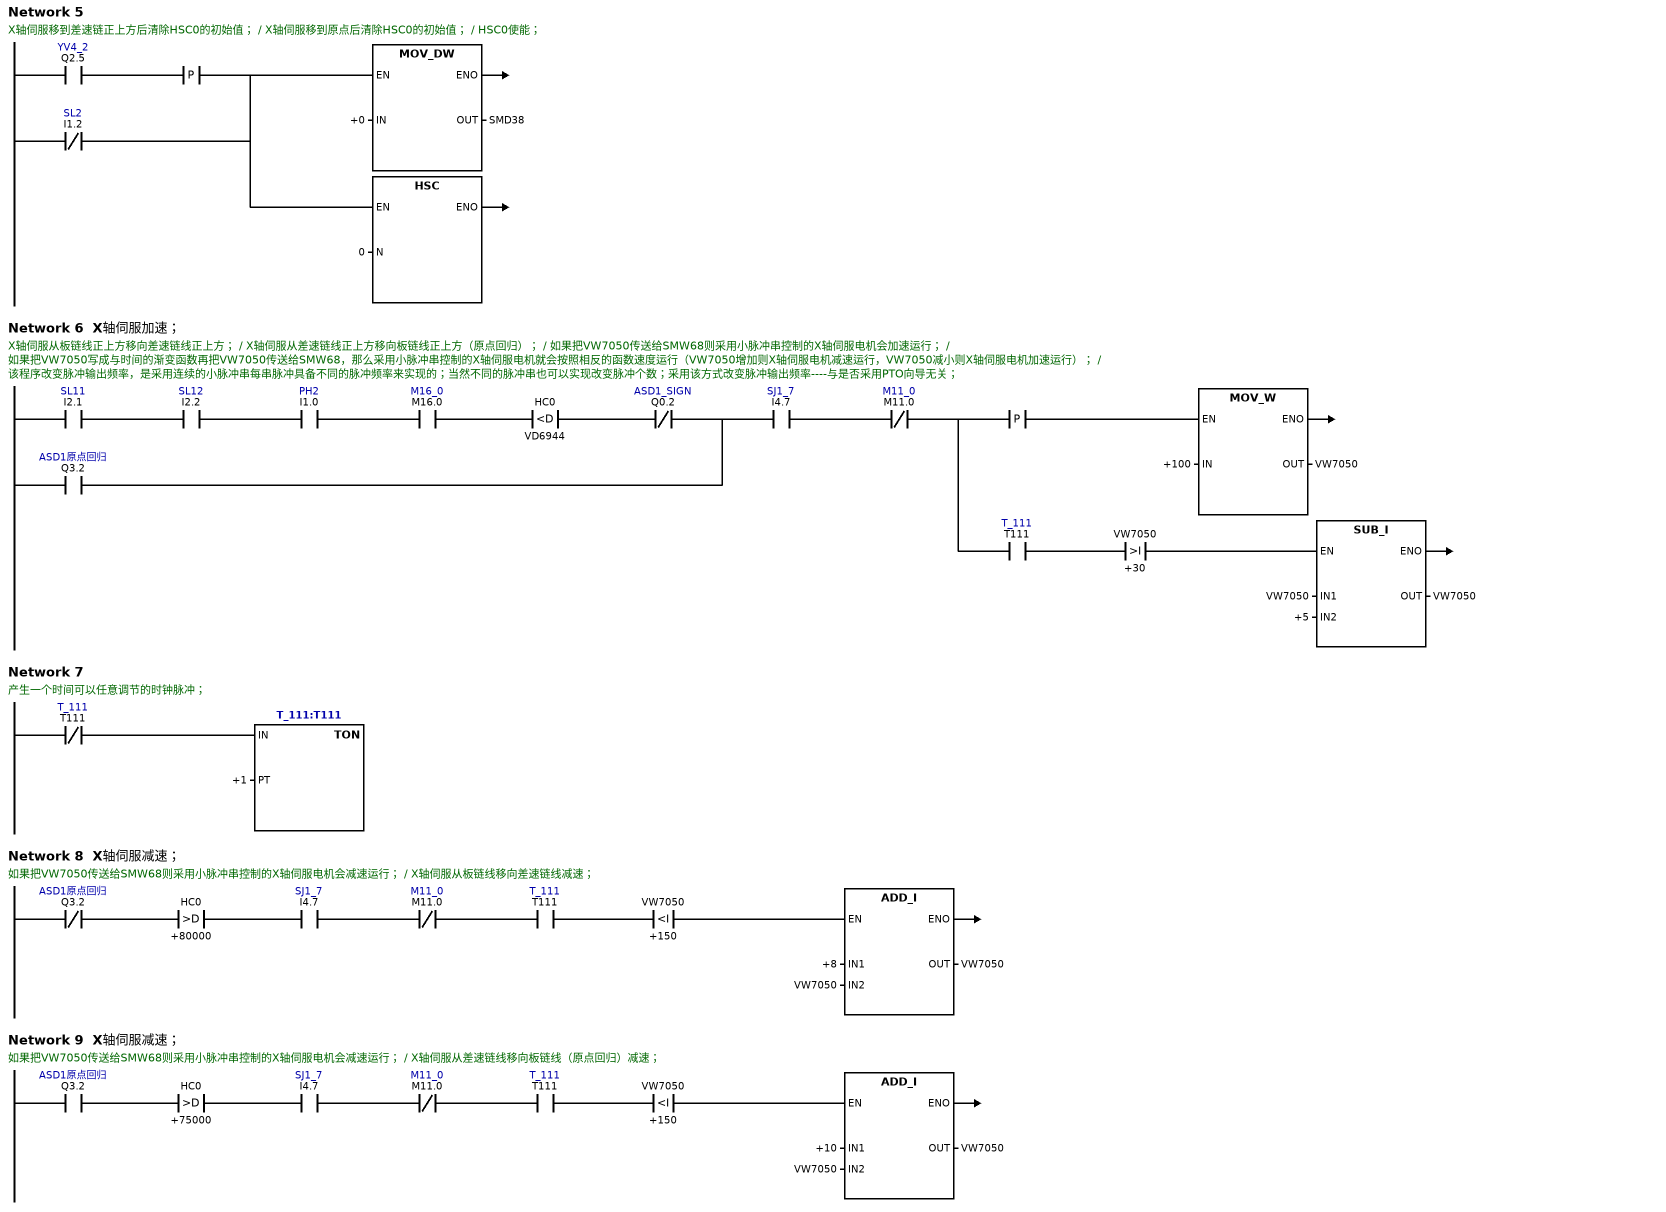
[picture p24: SBR11 networks 5-9]
Network 5
// X轴伺服移到差速链正上方后清除HSC0的初始值；
// X轴伺服移到原点后清除HSC0的初始值；
// HSC0使能；
LD     YV4_2:Q2.5
EU
ON     SL2:I1.2
MOVD   +0, SMD38
HSC    0
Network 6 // X轴伺服加速；
// X轴伺服从板链线正上方移向差速链线正上方；
// X轴伺服从差速链线正上方移向板链线正上方（原点回归）；
// 如果把VW7050传送给SMW68则采用小脉冲串控制的X轴伺服电机会加速运行；
// 如果把VW7050写成与时间的渐变函数再把VW7050传送给SMW68，那么采用小脉冲串控制的X轴伺服电机就会按照相反的函数速度运行（VW7050增加则X轴伺服电机减速运行，VW7050减小则X轴伺服电机加速运行）；
// 该程序改变脉冲输出频率，是采用连续的小脉冲串每串脉冲具备不同的脉冲频率来实现的；当然不同的脉冲串也可以实现改变脉冲个数；采用该方式改变脉冲输出频率----与是否采用PTO向导无关；
LD     SL11:I2.1
A      SL12:I2.2
A      PH2:I1.0
A      M16_0:M16.0
AD<    HC0, VD6944
AN     ASD1_SIGN:Q0.2
O      ASD1原点回归:Q3.2
A      SJ1_7:I4.7
AN     M11_0:M11.0
LPS
EU
MOVW   +100, VW7050
LPP
A      T_111:T111
AW>    VW7050, +30
-I     +5, VW7050
Network 7
// 产生一个时间可以任意调节的时钟脉冲；
LDN    T_111:T111
TON    T_111:T111, +1
Network 8 // X轴伺服减速；
// 如果把VW7050传送给SMW68则采用小脉冲串控制的X轴伺服电机会减速运行；
// X轴伺服从板链线移向差速链线减速；
LDN    ASD1原点回归:Q3.2
AD>    HC0, +80000
A      SJ1_7:I4.7
AN     M11_0:M11.0
A      T_111:T111
AW<    VW7050, +150
+I     +8, VW7050
Network 9 // X轴伺服减速；
// 如果把VW7050传送给SMW68则采用小脉冲串控制的X轴伺服电机会减速运行；
// X轴伺服从差速链线移向板链线（原点回归）减速；
LD     ASD1原点回归:Q3.2
AD>    HC0, +75000
A      SJ1_7:I4.7
AN     M11_0:M11.0
A      T_111:T111
AW<    VW7050, +150
+I     +10, VW7050
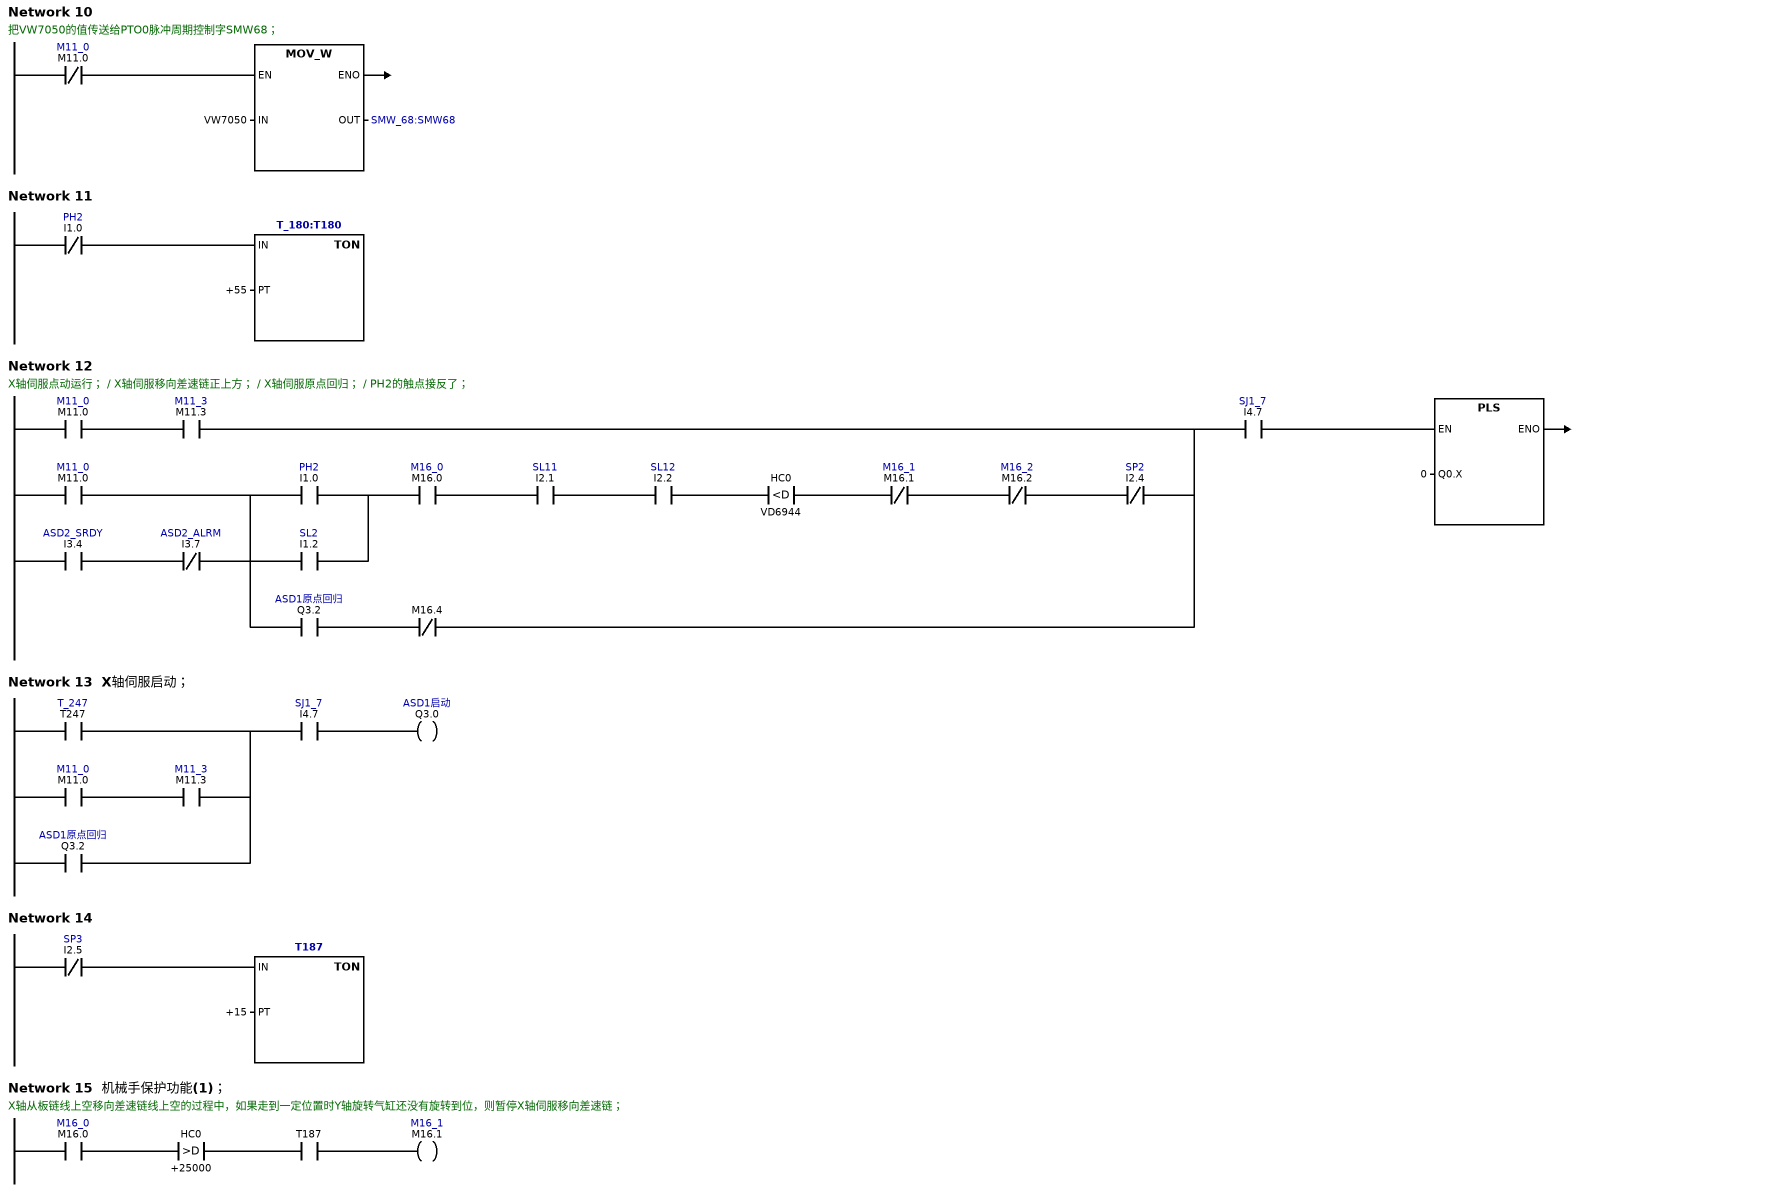
Network 10
// 把VW7050的值传送给PTO0脉冲周期控制字SMW68；
LDN    M11_0:M11.0
MOVW   VW7050, SMW_68:SMW68
Network 11
LDN    PH2:I1.0
TON    T_180:T180, +55
Network 12
// X轴伺服点动运行；
// X轴伺服移向差速链正上方；
// X轴伺服原点回归；
// PH2的触点接反了；
LD     M11_0:M11.0
A      M11_3:M11.3
LD     M11_0:M11.0
LD     ASD2_SRDY:I3.4
AN     ASD2_ALRM:I3.7
OLD
LD     PH2:I1.0
O      SL2:I1.2
A      M16_0:M16.0
A      SL11:I2.1
A      SL12:I2.2
AD<    HC0, VD6944
AN     M16_1:M16.1
AN     M16_2:M16.2
AN     SP2:I2.4
LD     ASD1原点回归:Q3.2
AN     M16.4
OLD
ALD
OLD
A      SJ1_7:I4.7
PLS    0
Network 13 // X轴伺服启动；
LD     T_247:T247
LD     M11_0:M11.0
A      M11_3:M11.3
OLD
O      ASD1原点回归:Q3.2
A      SJ1_7:I4.7
=      ASD1启动:Q3.0
Network 14
LDN    SP3:I2.5
TON    T187, +15
Network 15 // 机械手保护功能(1)；
// X轴从板链线上空移向差速链线上空的过程中，如果走到一定位置时Y轴旋转气缸还没有旋转到位，则暂停X轴伺服移向差速链；
LD     M16_0:M16.0
AD>    HC0, +25000
A      T187
=      M16_1:M16.1
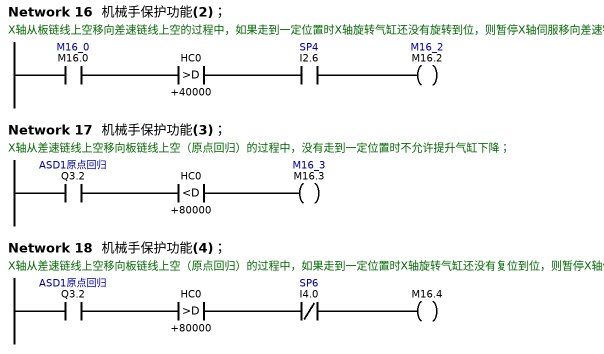
Network 16 // 机械手保护功能(2)；
// X轴从板链线上空移向差速链线上空的过程中，如果走到一定位置时X轴旋转气缸还没有旋转到位，则暂停X轴伺服移向差速链；
LD     M16_0:M16.0
AD>    HC0, +40000
A      SP4:I2.6
=      M16_2:M16.2
Network 17 // 机械手保护功能(3)；
// X轴从差速链线上空移向板链线上空（原点回归）的过程中，没有走到一定位置时不允许提升气缸下降；
LD     ASD1原点回归:Q3.2
AD<    HC0, +80000
=      M16_3:M16.3
Network 18 // 机械手保护功能(4)；
// X轴从差速链线上空移向板链线上空（原点回归）的过程中，如果走到一定位置时X轴旋转气缸还没有复位到位，则暂停X轴伺服移向板链线；
LD     ASD1原点回归:Q3.2
AD>    HC0, +80000
AN     SP6:I4.0
=      M16.4
END_SUBROUTINE_BLOCK

SUBROUTINE_BLOCK 机械手Y轴伺服控制:SBR12
TITLE=S7-200控制台达伺服电机----机械手Y轴伺服运动控制；
// 与X轴伺服控制类同；
BEGIN
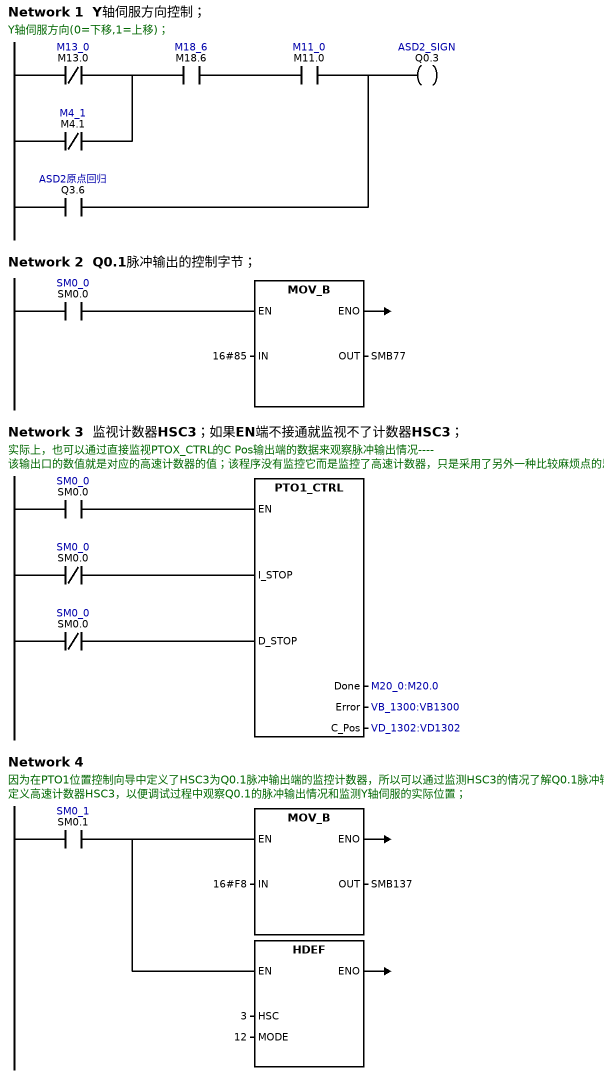
Network 1 // Y轴伺服方向控制；
// Y轴伺服方向(0=下移,1=上移)；
LDN    M13_0:M13.0
ON     M4_1:M4.1
A      M18_6:M18.6
A      M11_0:M11.0
O      ASD2原点回归:Q3.6
=      ASD2_SIGN:Q0.3
Network 2 // Q0.1脉冲输出的控制字节；
LD     SM0_0:SM0.0
MOVB   16#85, SMB77
Network 3 // 监视计数器HSC3；如果EN端不接通就监视不了计数器HSC3；
// 实际上，也可以通过直接监视PTOX_CTRL的C Pos输出端的数据来观察脉冲输出情况----该输出口的数值就是对应的高速计数器的值；该程序没有监控它而是监控了高速计数器，只是采用了另外一种比较麻烦点的思路而已，不建议采用；
LD     SM0_0:SM0.0
=      L60.0
LDN    SM0_0:SM0.0
=      L63.7
LDN    SM0_0:SM0.0
=      L63.6
LD     L60.0
CALL   PTO1_CTRL:SBR23, L63.7, L63.6, M20_0:M20.0, VB_1300:VB1300, VD_1302:VD1302
Network 4
// 因为在PTO1位置控制向导中定义了HSC3为Q0.1脉冲输出端的监控计数器，所以可以通过监测HSC3的情况了解Q0.1脉冲输出情况和监测Y轴伺服的实际位置；
// 定义高速计数器HSC3，以便调试过程中观察Q0.1的脉冲输出情况和监测Y轴伺服的实际位置；
LD     SM0_1:SM0.1
MOVB   16#F8, SMB137
HDEF   3, 12
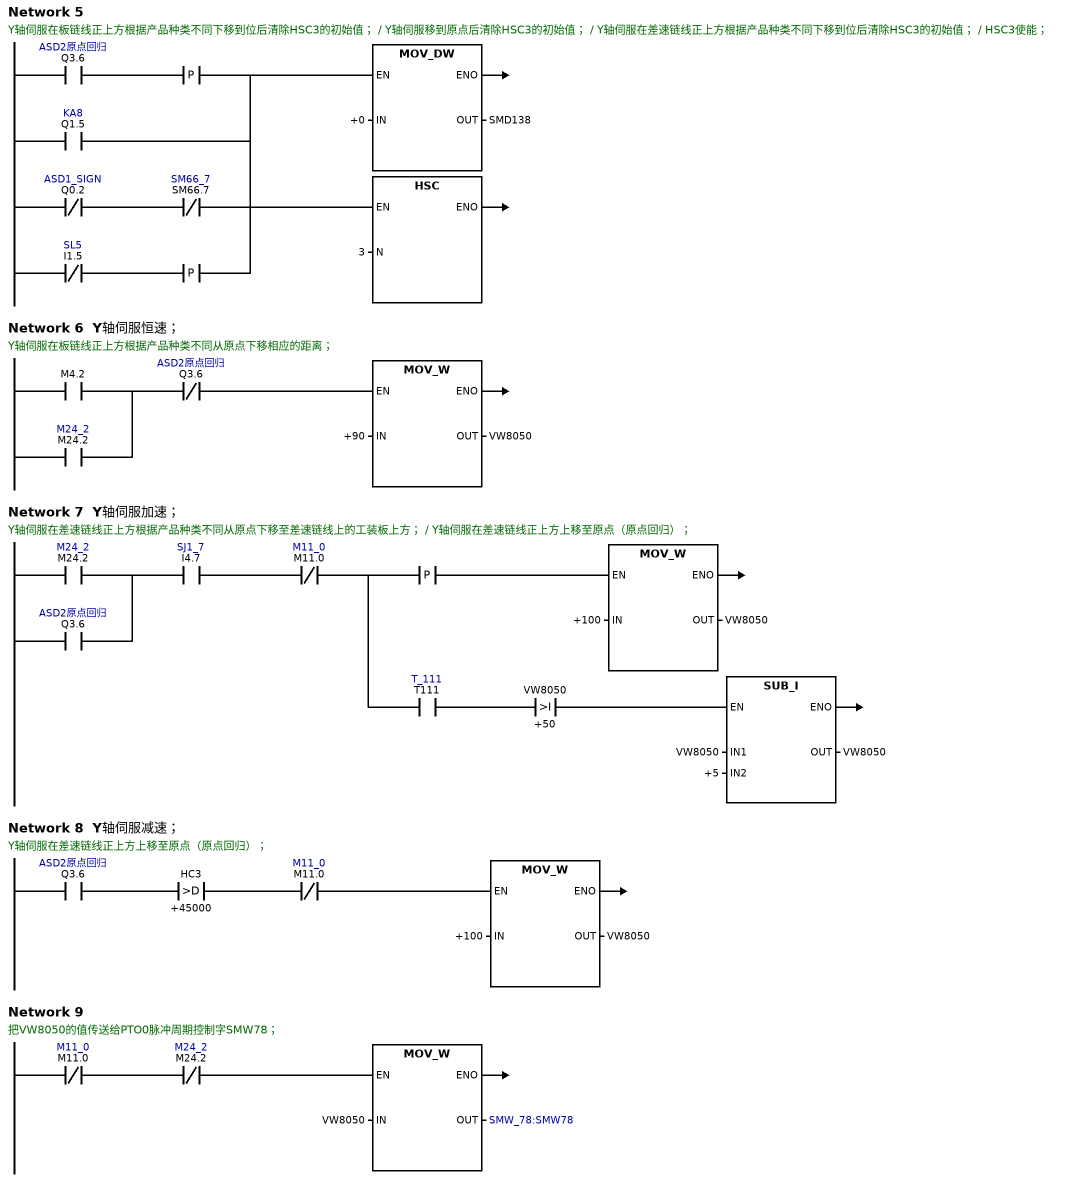
Network 5
// Y轴伺服在板链线正上方根据产品种类不同下移到位后清除HSC3的初始值；
// Y轴伺服移到原点后清除HSC3的初始值；
// Y轴伺服在差速链线正上方根据产品种类不同下移到位后清除HSC3的初始值；
// HSC3使能；
LD     ASD2原点回归:Q3.6
EU
O      KA8:Q1.5
LDN    ASD1_SIGN:Q0.2
AN     SM66_7:SM66.7
OLD
LDN    SL5:I1.5
EU
OLD
MOVD   +0, SMD138
HSC    3
Network 6 // Y轴伺服恒速；
// Y轴伺服在板链线正上方根据产品种类不同从原点下移相应的距离；
LD     M4.2
O      M24_2:M24.2
AN     ASD2原点回归:Q3.6
MOVW   +90, VW8050
Network 7 // Y轴伺服加速；
// Y轴伺服在差速链线正上方根据产品种类不同从原点下移至差速链线上的工装板上方；
// Y轴伺服在差速链线正上方上移至原点（原点回归）；
LD     M24_2:M24.2
O      ASD2原点回归:Q3.6
A      SJ1_7:I4.7
AN     M11_0:M11.0
LPS
EU
MOVW   +100, VW8050
LPP
A      T_111:T111
AW>    VW8050, +50
-I     +5, VW8050
Network 8 // Y轴伺服减速；
// Y轴伺服在差速链线正上方上移至原点（原点回归）；
LD     ASD2原点回归:Q3.6
AD>    HC3, +45000
AN     M11_0:M11.0
MOVW   +100, VW8050
Network 9
// 把VW8050的值传送给PTO0脉冲周期控制字SMW78；
LDN    M11_0:M11.0
AN     M24_2:M24.2
MOVW   VW8050, SMW_78:SMW78
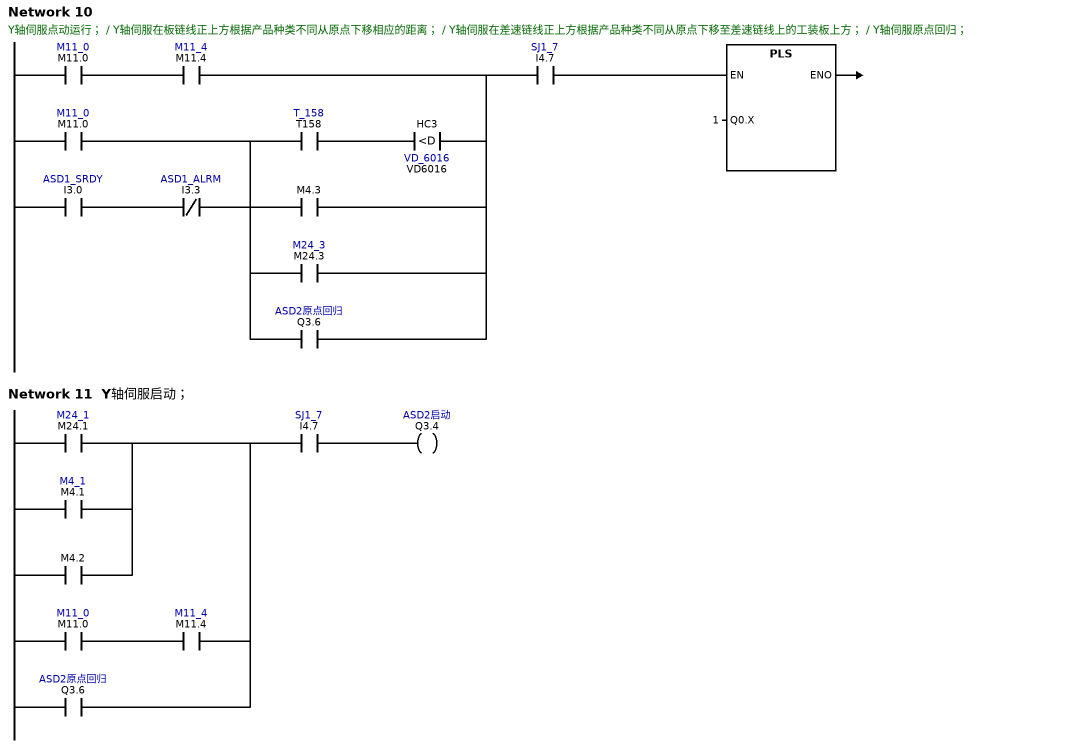
Network 10
// Y轴伺服点动运行；
// Y轴伺服在板链线正上方根据产品种类不同从原点下移相应的距离；
// Y轴伺服在差速链线正上方根据产品种类不同从原点下移至差速链线上的工装板上方；
// Y轴伺服原点回归；
LD     M11_0:M11.0
A      M11_4:M11.4
LD     M11_0:M11.0
LD     ASD1_SRDY:I3.0
AN     ASD1_ALRM:I3.3
OLD
LD     T_158:T158
AD<    HC3, VD_6016:VD6016
O      M4.3
O      M24_3:M24.3
O      ASD2原点回归:Q3.6
ALD
OLD
A      SJ1_7:I4.7
PLS    1
Network 11 // Y轴伺服启动；
LD     M24_1:M24.1
O      M4_1:M4.1
O      M4.2
LD     M11_0:M11.0
A      M11_4:M11.4
OLD
O      ASD2原点回归:Q3.6
A      SJ1_7:I4.7
=      ASD2启动:Q3.4
Network 16 // 网络标题
// 网络注释
END_SUBROUTINE_BLOCK

// SBR21: protected block, not included

// SBR22: protected block, not included

// SBR23: protected block, not included

// SBR24: protected block, not included

// (further data pages could not be read)
